ABB RobotStudio station: Coomportamiento1.rspag

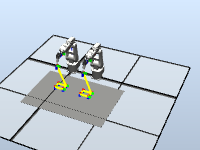
--- station ---
Station Coomportamiento1 (saved by RobotStudio 6.8.8307.1040)
Controller Sistema1, task T_ROB1: task frame (RAPID world) sits at (0, 502.68, 0) mm in the station
Controller IRB_120_3kg_0.58m
  mechanical unit ROB_1: IRB120_izda, 6 joints, base frame (0, 0, 0) mm
Controller Sistema1
  mechanical unit ROB_1: IRB120_dcha, 6 joints, base frame (0, 0, 0) mm
Layout (positions relative to the parent item):
  - IRB120_izda [mechanism, from Robots\IRB120_3_58_G_01.rslib] at (0, 0, 0) mm; joint values [0, 0, 0, 0, 0.5236, 0] (rad or m)
  - MyTool_izda [mechanism, from Training Objects\myTool.rslib] at (364.35, 0, 594) mm, rotated rx 180 ry 60 rz 180 deg
  - IRB120_dcha [mechanism, from Robots\IRB120_3_58_G_01.rslib] at (0, 502.68, 0) mm; joint values [0, 0, 0, 0, 0.5236, 0] (rad or m)
  - MyTool_dcha [mechanism, from Training Objects\myTool.rslib] at (364.35, 502.68, 594) mm, rotated rx 180 ry 60 rz 180 deg
  - mesa [part] at (187.06, -379.73, 0) mm
Attachment: MyTool_izda is attached to IRB120_izda / Link6
Attachment: MyTool_dcha is attached to IRB120_dcha / Link6

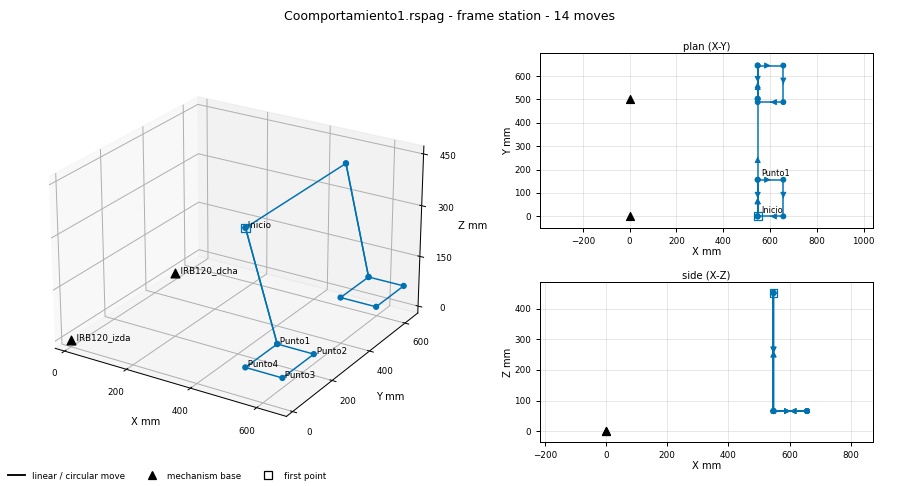
[picture p0: tool path of Coomportamiento1.rspag in frame station, 14 of 14 moves have a stored position in this frame; points joined in program order, loops and branches not executed]
--- Backups/IRB_120_3kg_0.58m/RAPID/TASK1/PROGMOD/CalibData.mod ---
MODULE CalibData
	PERS tooldata MyTool:=[TRUE,[[31.792631019,0,229.638935148],[0.945518576,0,0.325568154,0]],[1,[0,0,1],[1,0,0,0],0,0,0]];
ENDMODULE

--- Backups/IRB_120_3kg_0.58m/RAPID/TASK1/PROGMOD/Module1.mod ---
MODULE Module1
	CONST robtarget Inicio:=[[547.33065187,0,451.647288113],[0.19080896,0,0.98162719,0],[0,0,0,0],[9E+09,9E+09,9E+09,9E+09,9E+09,9E+09]];
	CONST robtarget Punto1:=[[547.330692564,156.503598902,65.645213658],[0.075178375,0.201157174,-0.97575764,0.042202269],[0,0,-1,0],[9E+09,9E+09,9E+09,9E+09,9E+09,9E+09]];
	CONST robtarget Punto2:=[[656.973912948,156.503608978,65.645121967],[0.075178434,0.201157179,-0.975757634,0.04220228],[0,0,-1,0],[9E+09,9E+09,9E+09,9E+09,9E+09,9E+09]];
	CONST robtarget Punto3:=[[656.974,0,65.645],[0.07517703,0.201160099,-0.975757176,0.042201449],[0,0,-1,0],[9E+09,9E+09,9E+09,9E+09,9E+09,9E+09]];
	CONST robtarget Punto4:=[[547.331,0,65.645],[0.07517703,0.201160099,-0.975757176,0.042201449],[0,0,-1,0],[9E+09,9E+09,9E+09,9E+09,9E+09,9E+09]];
    !***********************************************************
    !
    ! Módulo:  Module1
    !
    ! Descripción:
    !   <Introduzca la descripción aquí>
    !
    ! Autor: Nicolás
    !
    ! Versión: 1.0
    !
    !***********************************************************


    !***********************************************************
    !
    ! Procedimiento Main
    !
    !   Este es el punto de entrada de su programa
    !
    !***********************************************************
    PROC main()
        !Añada aquí su código
        Path_10;
    ENDPROC
	PROC Path_10()
	    MoveL Inicio,v50,fine,MyTool\WObj:=wobj0;
	    MoveL Punto1,v50,fine,MyTool\WObj:=wobj0;
	    MoveL Punto2,v50,fine,MyTool\WObj:=wobj0;
	    MoveL Punto3,v50,fine,MyTool\WObj:=wobj0;
	    MoveL Punto4,v50,fine,MyTool\WObj:=wobj0;
	    MoveL Punto1,v50,fine,MyTool\WObj:=wobj0;
	    MoveL Inicio,v50,fine,MyTool\WObj:=wobj0;
	ENDPROC
ENDMODULE

--- Backups/Sistema1/RAPID/TASK1/PROGMOD/Module1.mod ---
MODULE Module1
	CONST robtarget Inicio:=[[547.330665099,0,451.64730631],[0.190808996,0,0.981627183,0],[0,0,0,0],[9E+09,9E+09,9E+09,9E+09,9E+09,9E+09]];
	CONST robtarget Punto1:=[[547.331,142.188282773,65.65],[0.03960402,0.040733963,-0.994292869,0.090299267],[0,-1,0,0],[9E+09,9E+09,9E+09,9E+09,9E+09,9E+09]];
	CONST robtarget Punto2:=[[656.974,142.188282773,65.65],[0.03960402,0.040733963,-0.994292869,0.090299267],[0,-1,0,0],[9E+09,9E+09,9E+09,9E+09,9E+09,9E+09]];
	CONST robtarget Punto3:=[[656.974,-14.315717227,65.65],[0.03960402,0.040733963,-0.994292869,0.090299267],[0,-1,0,0],[9E+09,9E+09,9E+09,9E+09,9E+09,9E+09]];
	CONST robtarget Punto4:=[[547.331,-14.315717227,65.65],[0.03960402,0.040733963,-0.994292869,0.090299267],[0,-1,0,0],[9E+09,9E+09,9E+09,9E+09,9E+09,9E+09]];
    !***********************************************************
    !
    ! Módulo:  Module1
    !
    ! Descripción:
    !   <Introduzca la descripción aquí>
    !
    ! Autor: Nicolás
    !
    ! Versión: 1.0
    !
    !***********************************************************


    !***********************************************************
    !
    ! Procedimiento Main
    !
    !   Este es el punto de entrada de su programa
    !
    !***********************************************************
    PROC main()
        !Añada aquí su código
        Path_10;
    ENDPROC
	PROC Path_10()
	    MoveL Inicio,v50,fine,MyTool\WObj:=wobj0;
	    MoveL Punto1,v50,fine,MyTool\WObj:=wobj0;
	    MoveL Punto2,v50,fine,MyTool\WObj:=wobj0;
	    MoveL Punto3,v50,fine,MyTool\WObj:=wobj0;
	    MoveL Punto4,v50,fine,MyTool\WObj:=wobj0;
	    MoveL Punto1,v50,fine,MyTool\WObj:=wobj0;
	    MoveL Inicio,v50,fine,MyTool\WObj:=wobj0;
	ENDPROC
ENDMODULE
